// TIA Portal project "SWNC MK2" (V16)

(* hardware
DEVICE "S7-1200 station_1"  S7-1200 Station
   slot 0: "Rack_0"  S7-1200 Rack  Rack  V1.0
   slot 1: "RSF_PLC_Rupert"  CPU 1214C DC/DC/DC  6ES7 214-1AG40-0XB0  V4.4
   slot 2: "DI 8x24VDC_1"  6ES7 221-1BF32-0XB0  V2.0
   slot 3: "CB 1241 (RS485)"  CB 1241 (RS485)  6ES7 241-1CH30-1XB0  V1.0
   slot 3: "DQ 8xRelay_1"  SM 1222 DQ8 x relay  6ES7 222-1HF32-0XB0  V2.0
   slot 4: "AI 8x13BIT_1"  6ES7 231-4HF32-0XB0  V2.1
   slot 5: "AQ 2x14BIT_1"  SM 1232 AQ2  6ES7 232-4HB32-0XB0  V2.1
*)

// ===== PLC "RSF_PLC_Rupert"  CPU 1214C DC/DC/DC =====

VAR_GLOBAL   // PLC tag table "Default tag table"
   "System_Byte" AT %MB1000 : Byte;
   "FirstScan" AT %M1000.0 : Bool;
   "DiagStatusUpdate" AT %M1000.1 : Bool;
   "AlwaysTRUE" AT %M1000.2 : Bool;
   "AlwaysFALSE" AT %M1000.3 : Bool;
   "Clock_Byte" AT %MB1001 : Byte;
   "Clock_10Hz" AT %M1001.0 : Bool;
   "Clock_5Hz" AT %M1001.1 : Bool;
   "Clock_2.5Hz" AT %M1001.2 : Bool;
   "Clock_2Hz" AT %M1001.3 : Bool;
   "Clock_1.25Hz" AT %M1001.4 : Bool;
   "Clock_1Hz" AT %M1001.5 : Bool;
   "Clock_0.625Hz" AT %M1001.6 : Bool;
   "Clock_0.5Hz" AT %M1001.7 : Bool;
   "Mode Bit" AT %MB0 : USInt;
   "HOA Off" AT %M1.0 : Bool;
   "HOA Manual" AT %M1.1 : Bool;
   "HOA Auto Run" AT %M1.2 : Bool;
   "Outside Fan" AT %M1.3 : Bool;
   "Inside Fan" AT %M1.4 : Bool;
   "Outside Cooling" AT %M1.5 : Bool;
   "Inside Cooling" AT %M1.6 : Bool;
   "pump out supply" AT %M1.7 : Bool;
   "pump out Chiller" AT %M2.0 : Bool;
   "pump out inside tank" AT %M2.1 : Bool;
   "Pump out outside tank" AT %M2.2 : Bool;
   "pump out purge tank" AT %M2.3 : Bool;
   "pump chiller circulation" AT %M2.4 : Bool;
   "valve from supply" AT %M2.5 : Bool;   // 0 = to outdoor 1= to indoor
   "valve from chiller" AT %M2.6 : Bool;   // 0 = to outdoor 1= to indoor
   "valve from inside" AT %M2.7 : Bool;   // 0 = to purge 1= to chiller
   "valve from outside" AT %M3.0 : Bool;   // 0 = to purge 1= to chiller
   "chiller enable" AT %M3.1 : Bool;
   "SB OUTSIDE COOLING" AT %M3.2 : Bool;
   "SB INSIDE COOLING" AT %M3.3 : Bool;
   "SB pump out supply" AT %M3.4 : Bool;
   "SB pump out Chiller" AT %M3.5 : Bool;
   "SB pump out inside tank" AT %M3.6 : Bool;
   "SB Pump out outside tank" AT %M3.7 : Bool;
   "SB pump out purge tank" AT %M4.0 : Bool;
   "SB pump chiller circulation" AT %M4.1 : Bool;
   "SB valve from supply" AT %M4.2 : Bool;
   "SB valve from chiller" AT %M4.3 : Bool;
   "SB valve from inside" AT %M4.4 : Bool;
   "SB valve from outside" AT %M4.5 : Bool;
   "SB chiller enable" AT %M4.6 : Bool;
   "SB INSIDE FAN" AT %M4.7 : Bool;
   "SB OUTSIDE FAN" AT %M5.0 : Bool;
   "inside change bit" AT %M5.1 : Bool;   // true when tank change is in progress
   "PB_chill to regen trans" AT %M5.2 : Bool;
   "PB_regen to chill trans" AT %M5.3 : Bool;
END_VAR

VAR_GLOBAL   // PLC tag table "level sensors"
   "supply empty" AT %M0.0 : Bool;
   "chiller full" AT %M0.1 : Bool;
   "chiller empty" AT %M0.2 : Bool;
   "inside full" AT %M0.3 : Bool;
   "inside discharge" AT %M0.4 : Bool;
   "inside empty" AT %M0.5 : Bool;
   "outside full" AT %M0.6 : Bool;
   "outside discharge" AT %M0.7 : Bool;
   "outside empty" AT %M10.0 : Bool;
   "purge full" AT %M10.1 : Bool;
   "purge empty" AT %M10.2 : Bool;
END_VAR

DATA_BLOCK "System Properties"   // DB1
{ S7_Optimized_Access := 'TRUE' }
VERSION : 0.1
   VAR
      "Time" : Struct
         "Current Time" : Time_Of_Day;
         "Night time start" : Time_Of_Day := TOD#20:00:00;
         "Night time end" : Time_Of_Day := TOD#06:00:00;
         "is it day???" : Bool;   // 1 = day, 0 = night
      END_STRUCT;
      "Situation Bits" : Struct
         HOA : Int;
         "Day Run" : Bool;
         "Night Run" : Bool;
         "Day Tank Change" : Int;
         "Night Regen Complete" : Bool;
         "Day/Night Transition Bit" : Int;   // 0= no trans 1= day to night 2= night to day
         "regen or chill" : Int;   // 0 = chill , 1 = regen 3 = transition in progress
         "chilling to regen transition" : Bool;
         "regen to chilling transition" : Bool;
      END_STRUCT;
   END_VAR
BEGIN
END_DATA_BLOCK

DATA_BLOCK "Outputs"   // DB2
{ S7_Optimized_Access := 'TRUE' }
VERSION : 0.1
   VAR
      Fans : Struct
         "Inside Fan" : Bool;
         "Outside Fan" : Bool;
      END_STRUCT;
      "Cooling Pad Pumps" : Struct
         "Inside Cooling" : Bool;
         "Outside Cooling" : Bool;
      END_STRUCT;
      Pumps : Struct
         "From Supply Tank" : Bool;
         "From Chiller Tank" : Bool;
         "From Inside Tank" : Bool;
         "From Outside Tank" : Bool;
         "From Purge Tank" : Bool;
         "Chiller Recirculation" : Bool;
      END_STRUCT;
      Valves : Struct
         "From Supply" : Bool;   // 0= to outdoor, 1= to indoor
         "From Chiller" : Bool;   // 0= to outdoor, 1= to indoor
         "From Indoor" : Bool;   // 0= to Purge, 1= to Chiller
         "From Outdoor" : Bool;   // 0= to Purge, 1= to Chiller
      END_STRUCT;
      Chiller : Struct
         "Chiller Enable" : Bool;
      END_STRUCT;
   END_VAR
BEGIN
END_DATA_BLOCK

DATA_BLOCK "Alarm Conditions"   // DB3
{ S7_Optimized_Access := 'TRUE' }
VERSION : 0.1
   VAR
      "E Stop Pushed" : Bool;
      "Pump Over run" : Bool;
      "Alarm bit" : Bool;
      "Alarm Reset" : Bool;
   END_VAR
BEGIN
END_DATA_BLOCK

DATA_BLOCK "What Time is it?_DB"   // DB4
{ S7_Optimized_Access := 'TRUE' }
VERSION : 0.1
// stored: InstanceOfName What Time is it?
"What Time is it?"
BEGIN
END_DATA_BLOCK

DATA_BLOCK "What mode_DB"   // DB5
{ S7_Optimized_Access := 'TRUE' }
VERSION : 0.1
// stored: InstanceOfName What mode
"What mode"
BEGIN
END_DATA_BLOCK

DATA_BLOCK "Manual Mode_DB"   // DB6
{ S7_Optimized_Access := 'TRUE' }
VERSION : 0.1
// stored: InstanceOfName Manual Mode
"Manual Mode"
BEGIN
END_DATA_BLOCK

DATA_BLOCK "Day Operation_DB"   // DB7
{ S7_Optimized_Access := 'TRUE' }
VERSION : 0.1
// stored: InstanceOfName Day Operation
"Day Operation"
BEGIN
END_DATA_BLOCK

DATA_BLOCK "Night Operation_DB"   // DB8
{ S7_Optimized_Access := 'TRUE' }
VERSION : 0.1
// stored: InstanceOfName Night Operation
"Night Operation"
BEGIN
END_DATA_BLOCK

DATA_BLOCK "Tank check_DB"   // DB9
{ S7_Optimized_Access := 'TRUE' }
VERSION : 0.1
// stored: InstanceOfName Tank check
"Tank check"
BEGIN
END_DATA_BLOCK

DATA_BLOCK "inside tank switch_DB"   // DB11
{ S7_Optimized_Access := 'TRUE' }
VERSION : 0.1
// stored: InstanceOfName inside tank switch
"inside tank switch"
BEGIN
END_DATA_BLOCK

DATA_BLOCK "Auto Run Program_DB"   // DB12
{ S7_Optimized_Access := 'TRUE' }
VERSION : 0.1
// stored: InstanceOfName Auto Run Program
"Auto Run Program"
BEGIN
END_DATA_BLOCK

DATA_BLOCK "Day to Night change_DB"   // DB13
{ S7_Optimized_Access := 'TRUE' }
VERSION : 0.1
// stored: InstanceOfName Day to Night change
"Day to Night change"
BEGIN
END_DATA_BLOCK

DATA_BLOCK "Night to Day change_DB"   // DB14
{ S7_Optimized_Access := 'TRUE' }
VERSION : 0.1
// stored: InstanceOfName Night to Day change
"Night to Day change"
BEGIN
END_DATA_BLOCK

DATA_BLOCK "check for regen transitions_DB"   // DB18
{ S7_Optimized_Access := 'TRUE' }
VERSION : 0.1
// stored: InstanceOfName check for regen transitions
"check for regen transitions"
BEGIN
END_DATA_BLOCK

DATA_BLOCK "chilling to regeneration trans_DB"   // DB19
{ S7_Optimized_Access := 'TRUE' }
VERSION : 0.1
// stored: InstanceOfName chilling to regeneration trans
"chilling to regeneration trans"
BEGIN
END_DATA_BLOCK

DATA_BLOCK "regeneration to chilling trans_DB"   // DB21
{ S7_Optimized_Access := 'TRUE' }
VERSION : 0.1
// stored: InstanceOfName regeneration to chilling trans
"regeneration to chilling trans"
BEGIN
END_DATA_BLOCK

// folder: System blocks/Program resources

DATA_BLOCK "IEC_Timer_0_DB"   // DB10
{ S7_Optimized_Access := 'TRUE' }
AUTHOR : Simatic
FAMILY : IEC
NAME : IEC_TMR
VERSION : 1.0
// stored: InstanceOfName IEC_TIMER
"IEC_TIMER"
BEGIN
END_DATA_BLOCK

DATA_BLOCK "IEC_Timer_0_DB_1"   // DB15
{ S7_Optimized_Access := 'TRUE' }
AUTHOR : Simatic
FAMILY : IEC
NAME : IEC_TMR
VERSION : 1.0
// stored: InstanceOfName IEC_TIMER
"IEC_TIMER"
BEGIN
END_DATA_BLOCK

DATA_BLOCK "IEC_Timer_0_DB_2"   // DB16
{ S7_Optimized_Access := 'TRUE' }
AUTHOR : Simatic
FAMILY : IEC
NAME : IEC_TMR
VERSION : 1.0
// stored: InstanceOfName IEC_TIMER
"IEC_TIMER"
BEGIN
END_DATA_BLOCK

DATA_BLOCK "IEC_Timer_0_DB_3"   // DB17
{ S7_Optimized_Access := 'TRUE' }
AUTHOR : Simatic
FAMILY : IEC
NAME : IEC_TMR
VERSION : 1.0
// stored: InstanceOfName IEC_TIMER
"IEC_TIMER"
BEGIN
END_DATA_BLOCK

DATA_BLOCK "IEC_Timer_0_DB_4"   // DB20
{ S7_Optimized_Access := 'TRUE' }
AUTHOR : Simatic
FAMILY : IEC
NAME : IEC_TMR
VERSION : 1.0
// stored: InstanceOfName IEC_TIMER
"IEC_TIMER"
BEGIN
END_DATA_BLOCK

// folder: (top level)

FUNCTION_BLOCK "What Time is it?"   // FB1, FBD
{ S7_Optimized_Access := 'TRUE' }
VERSION : 0.1
   VAR
      temp1 : DTL;
      OS1 : Bool;
      OS2 : Bool;
      LTNE : Bool;
   END_VAR
   VAR_TEMP
      temp2 : Int;
   END_VAR
   VAR_TEMP   // added for the SCL form of the ladder/FBD networks
      _w1 : Bool;
      _w2 : Bool;
      _w3 : Bool;
   END_VAR
BEGIN

REGION Network 1
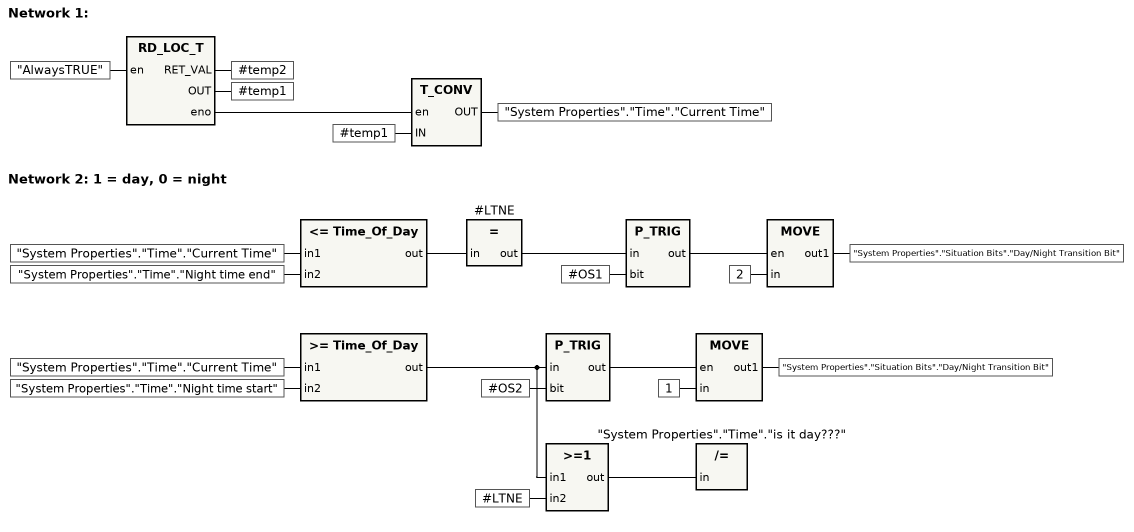
   // ENO of a box is taken as its EN; it also drops when the box reports an error
   #_w1 := "AlwaysTRUE";
   IF #_w1 THEN
       #temp2 := RD_LOC_T(OUT => #temp1);
       "System Properties"."Time"."Current Time" := T_CONV(IN := #temp1);
   END_IF;
END_REGION

REGION Network 2: 1 = day, 0 = night
   // also set the day/night transition integer
   // 0 = no transition
   // 1 = day to night transition
   // 2 = night to day transition
   #LTNE := "System Properties"."Time"."Current Time" <= "System Properties"."Time"."Night time end";
   #_w1 := #LTNE AND NOT #OS1;   // rising edge
   #OS1 := #LTNE;
   IF #_w1 THEN "System Properties"."Situation Bits"."Day/Night Transition Bit" := 2; END_IF;
   #_w2 := "System Properties"."Time"."Current Time" >= "System Properties"."Time"."Night time start";
   #_w3 := #_w2 AND NOT #OS2;   // rising edge
   #OS2 := #_w2;
   IF #_w3 THEN "System Properties"."Situation Bits"."Day/Night Transition Bit" := 1; END_IF;
   "System Properties"."Time"."is it day???" := NOT (#_w2 OR #LTNE);
END_REGION
END_FUNCTION_BLOCK

FUNCTION_BLOCK "What mode"   // FB2, LAD
{ S7_Optimized_Access := 'TRUE' }
VERSION : 0.1
BEGIN

REGION Network 1: Mode selection
   // 0 = startup
   // 1 = off
   // 2 = manual control
   // 3 = automatic run
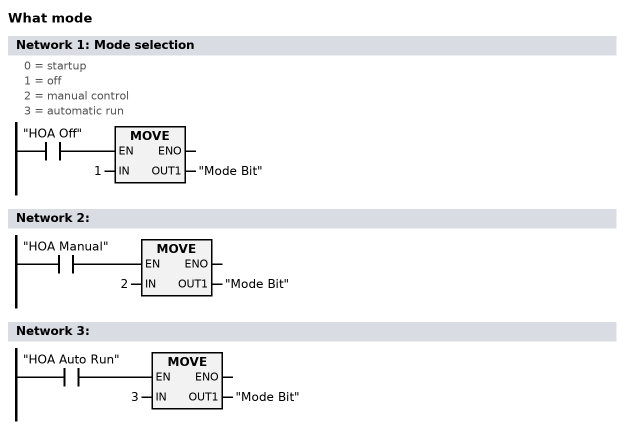
   RUNG wire#powerrail
      Contact( "HOA Off" )
      Move(in := 1, out1 => "Mode Bit")
   END_RUNG
   // the same network as SCL:
   IF "HOA Off" THEN "Mode Bit" := 1; END_IF;
END_REGION

REGION Network 2
   RUNG wire#powerrail
      Contact( "HOA Manual" )
      Move(in := 2, out1 => "Mode Bit")
   END_RUNG
   // the same network as SCL:
   IF "HOA Manual" THEN "Mode Bit" := 2; END_IF;
END_REGION

REGION Network 3
   RUNG wire#powerrail
      Contact( "HOA Auto Run" )
      Move(in := 3, out1 => "Mode Bit")
   END_RUNG
   // the same network as SCL:
   IF "HOA Auto Run" THEN "Mode Bit" := 3; END_IF;
END_REGION
END_FUNCTION_BLOCK

FUNCTION_BLOCK "Manual Mode"   // FB3, LAD
{ S7_Optimized_Access := 'TRUE' }
VERSION : 0.1
BEGIN

REGION Network 1: Manual operation of outputs
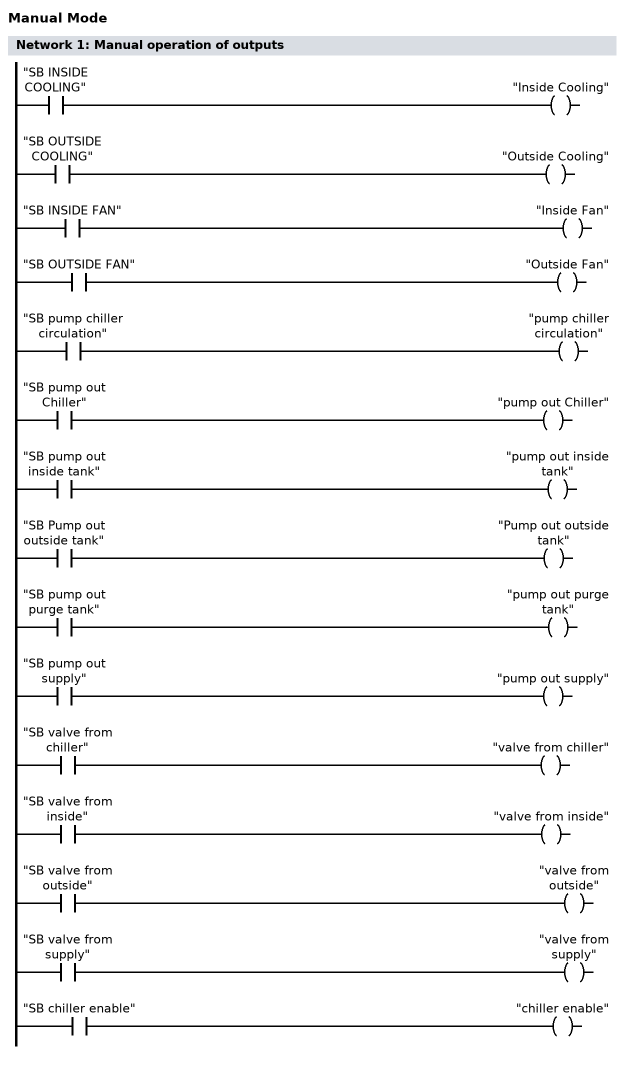
   RUNG wire#powerrail
      Contact( "SB INSIDE COOLING" )
      Coil( "Inside Cooling" )
   END_RUNG
   RUNG wire#powerrail
      Contact( "SB OUTSIDE COOLING" )
      Coil( "Outside Cooling" )
   END_RUNG
   RUNG wire#powerrail
      Contact( "SB INSIDE FAN" )
      Coil( "Inside Fan" )
   END_RUNG
   RUNG wire#powerrail
      Contact( "SB OUTSIDE FAN" )
      Coil( "Outside Fan" )
   END_RUNG
   RUNG wire#powerrail
      Contact( "SB pump chiller circulation" )
      Coil( "pump chiller circulation" )
   END_RUNG
   RUNG wire#powerrail
      Contact( "SB pump out Chiller" )
      Coil( "pump out Chiller" )
   END_RUNG
   RUNG wire#powerrail
      Contact( "SB pump out inside tank" )
      Coil( "pump out inside tank" )
   END_RUNG
   RUNG wire#powerrail
      Contact( "SB Pump out outside tank" )
      Coil( "Pump out outside tank" )
   END_RUNG
   RUNG wire#powerrail
      Contact( "SB pump out purge tank" )
      Coil( "pump out purge tank" )
   END_RUNG
   RUNG wire#powerrail
      Contact( "SB pump out supply" )
      Coil( "pump out supply" )
   END_RUNG
   RUNG wire#powerrail
      Contact( "SB valve from chiller" )
      Coil( "valve from chiller" )
   END_RUNG
   RUNG wire#powerrail
      Contact( "SB valve from inside" )
      Coil( "valve from inside" )
   END_RUNG
   RUNG wire#powerrail
      Contact( "SB valve from outside" )
      Coil( "valve from outside" )
   END_RUNG
   RUNG wire#powerrail
      Contact( "SB valve from supply" )
      Coil( "valve from supply" )
   END_RUNG
   RUNG wire#powerrail
      Contact( "SB chiller enable" )
      Coil( "chiller enable" )
   END_RUNG
   // the same network as SCL:
   "Inside Cooling" := "SB INSIDE COOLING";
   "Outside Cooling" := "SB OUTSIDE COOLING";
   "Inside Fan" := "SB INSIDE FAN";
   "Outside Fan" := "SB OUTSIDE FAN";
   "pump chiller circulation" := "SB pump chiller circulation";
   "pump out Chiller" := "SB pump out Chiller";
   "pump out inside tank" := "SB pump out inside tank";
   "Pump out outside tank" := "SB Pump out outside tank";
   "pump out purge tank" := "SB pump out purge tank";
   "pump out supply" := "SB pump out supply";
   "valve from chiller" := "SB valve from chiller";
   "valve from inside" := "SB valve from inside";
   "valve from outside" := "SB valve from outside";
   "valve from supply" := "SB valve from supply";
   "chiller enable" := "SB chiller enable";
END_REGION
END_FUNCTION_BLOCK

FUNCTION_BLOCK "Auto Run Program"   // FB4, LAD
{ S7_Optimized_Access := 'TRUE' }
VERSION : 0.1
BEGIN

REGION Network 1: Select for day or night operation
   // only works when there is not transitions happening
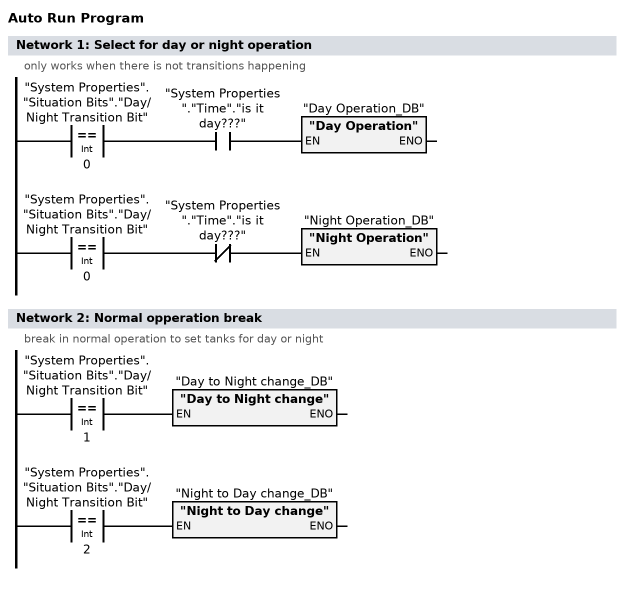
   RUNG wire#powerrail
      { S7_Templates := "SrcType := Int" } EQ_Contact(in1 := "System Properties"."Situation Bits"."Day/Night Transition Bit", in2 := 0)
      Contact( "System Properties"."Time"."is it day???" )
      "Day Operation_DB"()
   END_RUNG
   RUNG wire#powerrail
      { S7_Templates := "SrcType := Int" } EQ_Contact(in1 := "System Properties"."Situation Bits"."Day/Night Transition Bit", in2 := 0)
      I_Contact( "System Properties"."Time"."is it day???" )
      "Night Operation_DB"()
   END_RUNG
   // the same network as SCL:
   IF ("System Properties"."Situation Bits"."Day/Night Transition Bit" = 0) AND "System Properties"."Time"."is it day???" THEN
       "Day Operation_DB"();   // "Day Operation"
   END_IF;
   IF ("System Properties"."Situation Bits"."Day/Night Transition Bit" = 0) AND NOT "System Properties"."Time"."is it day???" THEN
       "Night Operation_DB"();   // "Night Operation"
   END_IF;
END_REGION

REGION Network 2: Normal opperation break
   // break in normal operation to set tanks for day or night
   RUNG wire#powerrail
      { S7_Templates := "SrcType := Int" } EQ_Contact(in1 := "System Properties"."Situation Bits"."Day/Night Transition Bit", in2 := 1)
      "Day to Night change_DB"()
   END_RUNG
   RUNG wire#powerrail
      { S7_Templates := "SrcType := Int" } EQ_Contact(in1 := "System Properties"."Situation Bits"."Day/Night Transition Bit", in2 := 2)
      "Night to Day change_DB"()
   END_RUNG
   // the same network as SCL:
   IF "System Properties"."Situation Bits"."Day/Night Transition Bit" = 1 THEN
       "Day to Night change_DB"();   // "Day to Night change"
   END_IF;
   IF "System Properties"."Situation Bits"."Day/Night Transition Bit" = 2 THEN
       "Night to Day change_DB"();   // "Night to Day change"
   END_IF;
END_REGION
END_FUNCTION_BLOCK

FUNCTION_BLOCK "Day Operation"   // FB5, LAD
{ S7_Optimized_Access := 'TRUE' }
VERSION : 0.1
   VAR_TEMP   // added for the SCL form of the ladder/FBD networks
      _w1 : Bool;
   END_VAR
BEGIN

REGION Network 1: Place Holder
   // to make VFD control
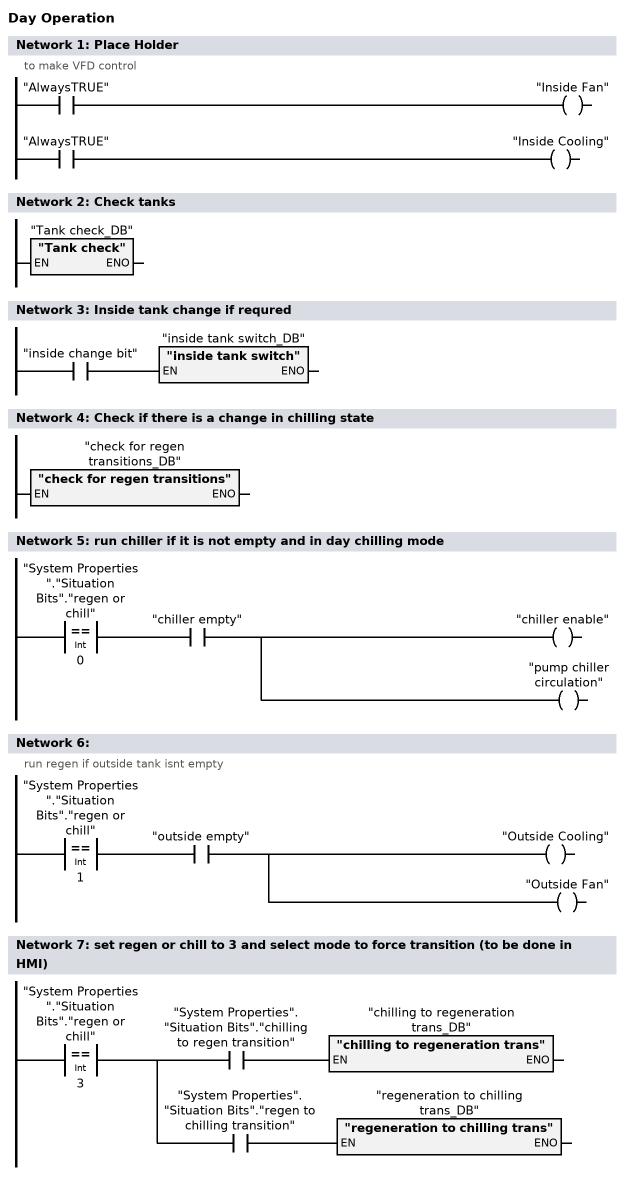
   RUNG wire#powerrail
      Contact( "AlwaysTRUE" )
      Coil( "Inside Fan" )
   END_RUNG
   RUNG wire#powerrail
      Contact( "AlwaysTRUE" )
      Coil( "Inside Cooling" )
   END_RUNG
   // the same network as SCL:
   "Inside Fan" := "AlwaysTRUE";
   "Inside Cooling" := "AlwaysTRUE";
END_REGION

REGION Network 2: Check tanks
   RUNG wire#powerrail
      "Tank check_DB"()
   END_RUNG
   // the same network as SCL:
   "Tank check_DB"();   // "Tank check"
END_REGION

REGION Network 3: Inside tank change if requred
   RUNG wire#powerrail
      Contact( "inside change bit" )
      "inside tank switch_DB"()
   END_RUNG
   // the same network as SCL:
   IF "inside change bit" THEN
       "inside tank switch_DB"();   // "inside tank switch"
   END_IF;
END_REGION

REGION Network 4: Check if there is a change in chilling state
   RUNG wire#powerrail
      "check for regen transitions_DB"()
   END_RUNG
   // the same network as SCL:
   "check for regen transitions_DB"();   // "check for regen transitions"
END_REGION

REGION Network 5: run chiller if it is not empty and in day chilling mode
   RUNG wire#powerrail
      { S7_Templates := "SrcType := Int" } EQ_Contact(in1 := "System Properties"."Situation Bits"."regen or chill", in2 := 0)
      Contact( "chiller empty" )
      wire#w1
      Coil( "chiller enable" )
   END_RUNG
   RUNG wire#w1
      Coil( "pump chiller circulation" )
   END_RUNG
   // the same network as SCL:
   "chiller enable" := ("System Properties"."Situation Bits"."regen or chill" = 0) AND "chiller empty";
   "pump chiller circulation" := "chiller enable";
END_REGION

REGION Network 6
   // run regen if outside tank isnt empty
   RUNG wire#powerrail
      { S7_Templates := "SrcType := Int" } EQ_Contact(in1 := "System Properties"."Situation Bits"."regen or chill", in2 := 1)
      Contact( "outside empty" )
      wire#w1
      Coil( "Outside Cooling" )
   END_RUNG
   RUNG wire#w1
      Coil( "Outside Fan" )
   END_RUNG
   // the same network as SCL:
   "Outside Cooling" := ("System Properties"."Situation Bits"."regen or chill" = 1) AND "outside empty";
   "Outside Fan" := "Outside Cooling";
END_REGION

REGION Network 7: set regen or chill to 3 and select mode to force transition (to be done in HMI)
   RUNG wire#powerrail
      { S7_Templates := "SrcType := Int" } EQ_Contact(in1 := "System Properties"."Situation Bits"."regen or chill", in2 := 3)
      wire#w1
      Contact( "System Properties"."Situation Bits"."chilling to regen transition" )
      "chilling to regeneration trans_DB"()
   END_RUNG
   RUNG wire#w1
      Contact( "System Properties"."Situation Bits"."regen to chilling transition" )
      "regeneration to chilling trans_DB"()
   END_RUNG
   // the same network as SCL:
   #_w1 := "System Properties"."Situation Bits"."regen or chill" = 3;
   IF #_w1 AND "System Properties"."Situation Bits"."chilling to regen transition" THEN
       "chilling to regeneration trans_DB"();   // "chilling to regeneration trans"
   END_IF;
   IF #_w1 AND "System Properties"."Situation Bits"."regen to chilling transition" THEN
       "regeneration to chilling trans_DB"();   // "regeneration to chilling trans"
   END_IF;
END_REGION
END_FUNCTION_BLOCK

FUNCTION_BLOCK "Night Operation"   // FB6, LAD
{ S7_Optimized_Access := 'TRUE' }
VERSION : 0.1
BEGIN

REGION Network 1
   // place holder will be VFD
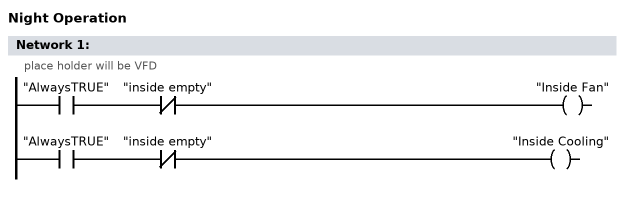
   RUNG wire#powerrail
      Contact( "AlwaysTRUE" )
      I_Contact( "inside empty" )
      Coil( "Inside Fan" )
   END_RUNG
   RUNG wire#powerrail
      Contact( "AlwaysTRUE" )
      I_Contact( "inside empty" )
      Coil( "Inside Cooling" )
   END_RUNG
   // the same network as SCL:
   "Inside Fan" := "AlwaysTRUE" AND NOT "inside empty";
   "Inside Cooling" := "AlwaysTRUE" AND NOT "inside empty";
END_REGION
END_FUNCTION_BLOCK

FUNCTION_BLOCK "Tank check"   // FB7, LAD
{ S7_Optimized_Access := 'TRUE' }
VERSION : 0.1
BEGIN

REGION Network 1: sets to true when the inside tank hits its discharge level
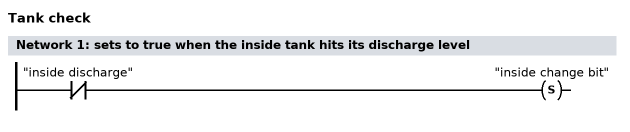
   RUNG wire#powerrail
      I_Contact( "inside discharge" )
      S_Coil( "inside change bit" )
   END_RUNG
   // the same network as SCL:
   IF NOT "inside discharge" THEN "inside change bit" := TRUE; END_IF;
END_REGION
END_FUNCTION_BLOCK

FUNCTION_BLOCK "inside tank switch"   // FB8, LAD
{ S7_Optimized_Access := 'TRUE' }
VERSION : 0.1
   VAR_TEMP   // added for the SCL form of the ladder/FBD networks
      _w1 : Bool;
   END_VAR
BEGIN

REGION Network 1: valve set up --- 0 = to purge 1= to chiller
   // set to purge (valve is not energised)
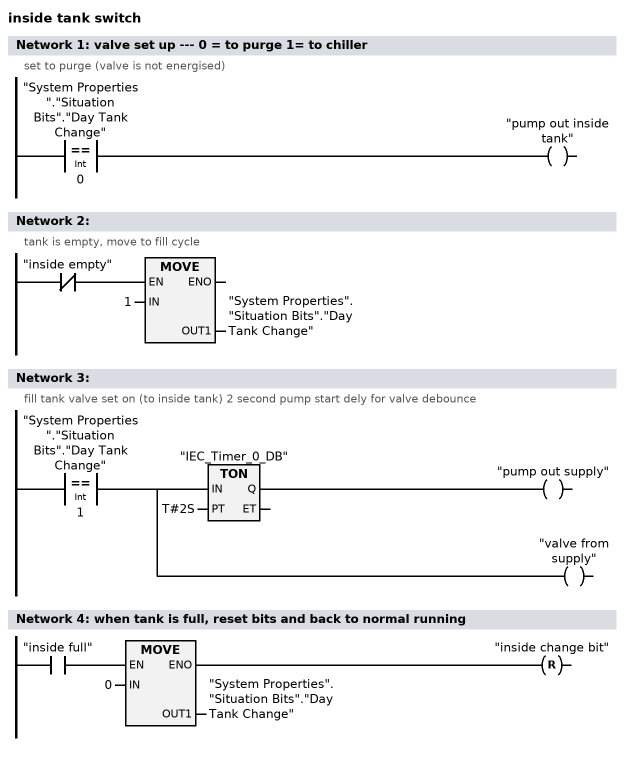
   RUNG wire#powerrail
      { S7_Templates := "SrcType := Int" } EQ_Contact(in1 := "System Properties"."Situation Bits"."Day Tank Change", in2 := 0)
      Coil( "pump out inside tank" )
   END_RUNG
   // the same network as SCL:
   "pump out inside tank" := "System Properties"."Situation Bits"."Day Tank Change" = 0;
END_REGION

REGION Network 2
   // tank is empty, move to fill cycle
   RUNG wire#powerrail
      I_Contact( "inside empty" )
      Move(in := 1, out1 => "System Properties"."Situation Bits"."Day Tank Change")
   END_RUNG
   // the same network as SCL:
   IF NOT "inside empty" THEN "System Properties"."Situation Bits"."Day Tank Change" := 1; END_IF;
END_REGION

REGION Network 3
   // fill tank valve set on (to inside tank) 2 second pump start dely for valve debounce
   #_w1 := "System Properties"."Situation Bits"."Day Tank Change" = 1;
   "IEC_Timer_0_DB".TON(IN := #_w1, PT := T#2S);
   "pump out supply" := "IEC_Timer_0_DB".Q;
   "valve from supply" := #_w1;
END_REGION

REGION Network 4: when tank is full, reset bits and back to normal running
   RUNG wire#powerrail
      Contact( "inside full" )
      Move(in := 0, out1 => "System Properties"."Situation Bits"."Day Tank Change")
      R_Coil( "inside change bit" )
   END_RUNG
   // the same network as SCL:
   IF "inside full" THEN
       "System Properties"."Situation Bits"."Day Tank Change" := 0;
       "inside change bit" := FALSE;
   END_IF;
END_REGION
END_FUNCTION_BLOCK

FUNCTION_BLOCK "Day to Night change"   // FB9, LAD
{ S7_Optimized_Access := 'TRUE' }
VERSION : 0.1
   VAR
      "DN change bit" : Int;
   END_VAR
   VAR_TEMP   // added for the SCL form of the ladder/FBD networks
      _w1 : Bool;
   END_VAR
BEGIN

REGION Network 1
   // inside tank to purge (valve at 0)
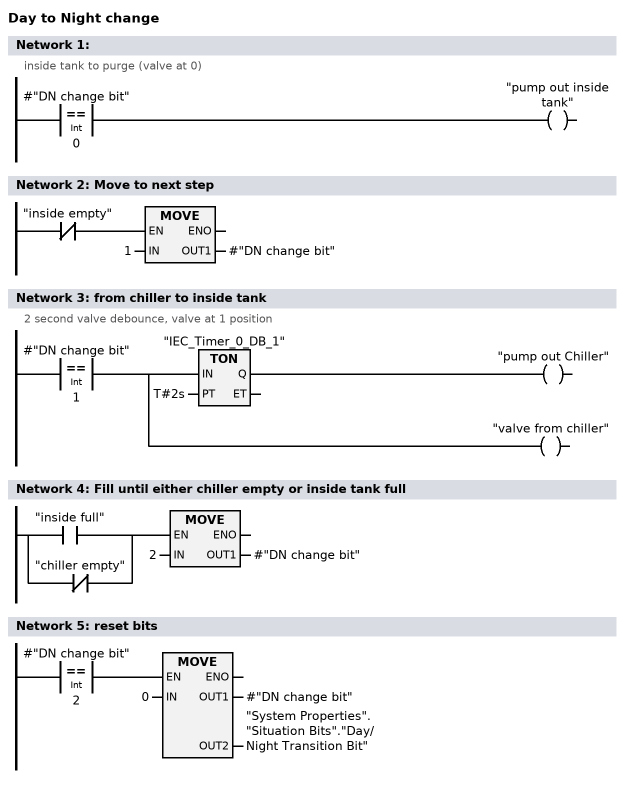
   RUNG wire#powerrail
      { S7_Templates := "SrcType := Int" } EQ_Contact(in1 := #"DN change bit", in2 := 0)
      Coil( "pump out inside tank" )
   END_RUNG
   // the same network as SCL:
   "pump out inside tank" := #"DN change bit" = 0;
END_REGION

REGION Network 2: Move to next step
   RUNG wire#powerrail
      I_Contact( "inside empty" )
      Move(in := 1, out1 => #"DN change bit")
   END_RUNG
   // the same network as SCL:
   IF NOT "inside empty" THEN #"DN change bit" := 1; END_IF;
END_REGION

REGION Network 3: from chiller to inside tank
   // 2 second valve debounce, valve at 1 position
   #_w1 := #"DN change bit" = 1;
   "IEC_Timer_0_DB_1".TON(IN := #_w1, PT := T#2s);
   "pump out Chiller" := "IEC_Timer_0_DB_1".Q;
   "valve from chiller" := #_w1;
END_REGION

REGION Network 4: Fill until either chiller empty or inside tank full
   RUNG wire#powerrail
      Contact( "inside full" )
      wire#w1
      Move(in := 2, out1 => #"DN change bit")
   END_RUNG
   RUNG wire#powerrail
      I_Contact( "chiller empty" )
   END_RUNG wire#w1
   // the same network as SCL:
   IF "inside full" OR NOT "chiller empty" THEN #"DN change bit" := 2; END_IF;
END_REGION

REGION Network 5: reset bits
   RUNG wire#powerrail
      { S7_Templates := "SrcType := Int" } EQ_Contact(in1 := #"DN change bit", in2 := 2)
      Move(in := 0, out1 => #"DN change bit", out2 => "System Properties"."Situation Bits"."Day/Night Transition Bit")
   END_RUNG
   // the same network as SCL:
   IF #"DN change bit" = 2 THEN
       #"DN change bit" := 0;
       "System Properties"."Situation Bits"."Day/Night Transition Bit" := 0;
   END_IF;
END_REGION
END_FUNCTION_BLOCK

FUNCTION_BLOCK "Night to Day change"   // FB10, LAD
{ S7_Optimized_Access := 'TRUE' }
VERSION : 0.1
   VAR
      "ND change bit" : Int;
   END_VAR
   VAR_TEMP   // added for the SCL form of the ladder/FBD networks
      _w1 : Bool;
   END_VAR
BEGIN

REGION Network 1: move from inside back to chiller
   // 2 second valve debounce
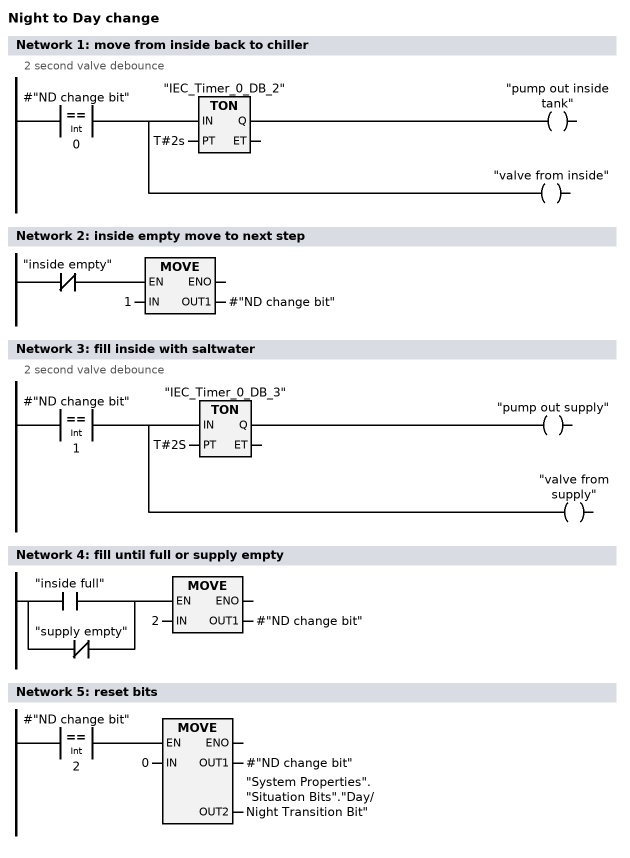
   #_w1 := #"ND change bit" = 0;
   "IEC_Timer_0_DB_2".TON(IN := #_w1, PT := T#2s);
   "pump out inside tank" := "IEC_Timer_0_DB_2".Q;
   "valve from inside" := #_w1;
END_REGION

REGION Network 2: inside empty move to next step
   RUNG wire#powerrail
      I_Contact( "inside empty" )
      Move(in := 1, out1 => #"ND change bit")
   END_RUNG
   // the same network as SCL:
   IF NOT "inside empty" THEN #"ND change bit" := 1; END_IF;
END_REGION

REGION Network 3: fill inside with saltwater
   // 2 second valve debounce
   #_w1 := #"ND change bit" = 1;
   "IEC_Timer_0_DB_3".TON(IN := #_w1, PT := T#2S);
   "pump out supply" := "IEC_Timer_0_DB_3".Q;
   "valve from supply" := #_w1;
END_REGION

REGION Network 4: fill until full or supply empty
   RUNG wire#powerrail
      Contact( "inside full" )
      wire#w1
      Move(in := 2, out1 => #"ND change bit")
   END_RUNG
   RUNG wire#powerrail
      I_Contact( "supply empty" )
   END_RUNG wire#w1
   // the same network as SCL:
   IF "inside full" OR NOT "supply empty" THEN #"ND change bit" := 2; END_IF;
END_REGION

REGION Network 5: reset bits
   RUNG wire#powerrail
      { S7_Templates := "SrcType := Int" } EQ_Contact(in1 := #"ND change bit", in2 := 2)
      Move(in := 0, out1 => #"ND change bit", out2 => "System Properties"."Situation Bits"."Day/Night Transition Bit")
   END_RUNG
   // the same network as SCL:
   IF #"ND change bit" = 2 THEN
       #"ND change bit" := 0;
       "System Properties"."Situation Bits"."Day/Night Transition Bit" := 0;
   END_IF;
END_REGION
END_FUNCTION_BLOCK

FUNCTION_BLOCK "check for regen transitions"   // FB11, LAD
{ S7_Optimized_Access := 'TRUE' }
VERSION : 0.1
   VAR
      OS3 : Bool;
      OS4 : Bool;
   END_VAR
   VAR_TEMP   // added for the SCL form of the ladder/FBD networks
      _w1 : Bool;
   END_VAR
BEGIN

REGION Network 1
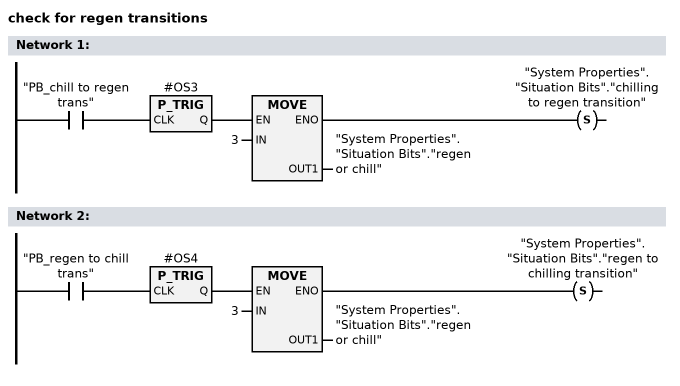
   RUNG wire#powerrail
      Contact( "PB_chill to regen trans" )
      P_Trig( #OS3 )
      Move(in := 3, out1 => "System Properties"."Situation Bits"."regen or chill")
      S_Coil( "System Properties"."Situation Bits"."chilling to regen transition" )
   END_RUNG
   // the same network as SCL:
   #_w1 := "PB_chill to regen trans" AND NOT #OS3;   // rising edge
   #OS3 := "PB_chill to regen trans";
   IF #_w1 THEN
       "System Properties"."Situation Bits"."regen or chill" := 3;
       "System Properties"."Situation Bits"."chilling to regen transition" := TRUE;
   END_IF;
END_REGION

REGION Network 2
   RUNG wire#powerrail
      Contact( "PB_regen to chill trans" )
      P_Trig( #OS4 )
      Move(in := 3, out1 => "System Properties"."Situation Bits"."regen or chill")
      S_Coil( "System Properties"."Situation Bits"."regen to chilling transition" )
   END_RUNG
   // the same network as SCL:
   #_w1 := "PB_regen to chill trans" AND NOT #OS4;   // rising edge
   #OS4 := "PB_regen to chill trans";
   IF #_w1 THEN
       "System Properties"."Situation Bits"."regen or chill" := 3;
       "System Properties"."Situation Bits"."regen to chilling transition" := TRUE;
   END_IF;
END_REGION
END_FUNCTION_BLOCK

FUNCTION_BLOCK "chilling to regeneration trans"   // FB12, LAD
{ S7_Optimized_Access := 'TRUE' }
VERSION : 0.1
   VAR
      "internal bit" : Int;
   END_VAR
   VAR_TEMP   // added for the SCL form of the ladder/FBD networks
      _w1 : Bool;
   END_VAR
BEGIN

REGION Network 1: make sure outside is empty
   // valve in position 0 to purge
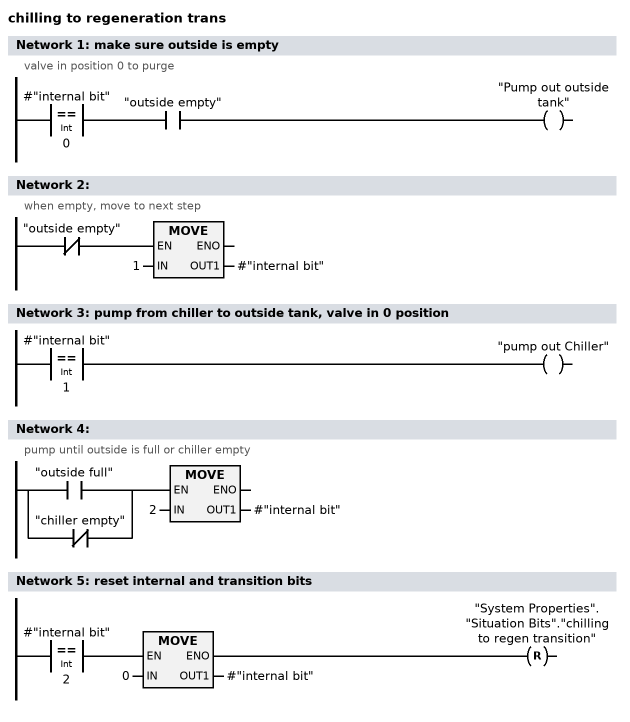
   RUNG wire#powerrail
      { S7_Templates := "SrcType := Int" } EQ_Contact(in1 := #"internal bit", in2 := 0)
      Contact( "outside empty" )
      Coil( "Pump out outside tank" )
   END_RUNG
   // the same network as SCL:
   "Pump out outside tank" := (#"internal bit" = 0) AND "outside empty";
END_REGION

REGION Network 2
   // when empty, move to next step
   RUNG wire#powerrail
      I_Contact( "outside empty" )
      Move(in := 1, out1 => #"internal bit")
   END_RUNG
   // the same network as SCL:
   IF NOT "outside empty" THEN #"internal bit" := 1; END_IF;
END_REGION

REGION Network 3: pump from chiller to outside tank, valve in 0 position
   RUNG wire#powerrail
      { S7_Templates := "SrcType := Int" } EQ_Contact(in1 := #"internal bit", in2 := 1)
      Coil( "pump out Chiller" )
   END_RUNG
   // the same network as SCL:
   "pump out Chiller" := #"internal bit" = 1;
END_REGION

REGION Network 4
   // pump until outside is full or chiller empty
   RUNG wire#powerrail
      Contact( "outside full" )
      wire#w1
      Move(in := 2, out1 => #"internal bit")
   END_RUNG
   RUNG wire#powerrail
      I_Contact( "chiller empty" )
   END_RUNG wire#w1
   // the same network as SCL:
   IF "outside full" OR NOT "chiller empty" THEN #"internal bit" := 2; END_IF;
END_REGION

REGION Network 5: reset internal and transition bits
   RUNG wire#powerrail
      { S7_Templates := "SrcType := Int" } EQ_Contact(in1 := #"internal bit", in2 := 2)
      Move(in := 0, out1 => #"internal bit")
      R_Coil( "System Properties"."Situation Bits"."chilling to regen transition" )
   END_RUNG
   // the same network as SCL:
   #_w1 := #"internal bit" = 2;
   IF #_w1 THEN
       #"internal bit" := 0;
       "System Properties"."Situation Bits"."chilling to regen transition" := FALSE;
   END_IF;
END_REGION
END_FUNCTION_BLOCK

FUNCTION_BLOCK "regeneration to chilling trans"   // FB13, LAD
{ S7_Optimized_Access := 'TRUE' }
VERSION : 0.1
   VAR
      "internal bit" : Int;
   END_VAR
   VAR_TEMP   // added for the SCL form of the ladder/FBD networks
      _w1 : Bool;
   END_VAR
BEGIN

REGION Network 1: empty outside tank to chiller
   // 2 second valve debounce
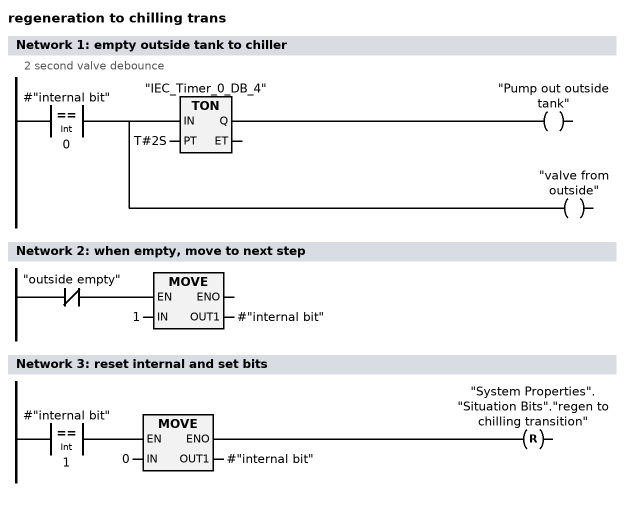
   #_w1 := #"internal bit" = 0;
   "IEC_Timer_0_DB_4".TON(IN := #_w1, PT := T#2S);
   "Pump out outside tank" := "IEC_Timer_0_DB_4".Q;
   "valve from outside" := #_w1;
END_REGION

REGION Network 2: when empty, move to next step
   RUNG wire#powerrail
      I_Contact( "outside empty" )
      Move(in := 1, out1 => #"internal bit")
   END_RUNG
   // the same network as SCL:
   IF NOT "outside empty" THEN #"internal bit" := 1; END_IF;
END_REGION

REGION Network 3: reset internal and set bits
   RUNG wire#powerrail
      { S7_Templates := "SrcType := Int" } EQ_Contact(in1 := #"internal bit", in2 := 1)
      Move(in := 0, out1 => #"internal bit")
      R_Coil( "System Properties"."Situation Bits"."regen to chilling transition" )
   END_RUNG
   // the same network as SCL:
   #_w1 := #"internal bit" = 1;
   IF #_w1 THEN
       #"internal bit" := 0;
       "System Properties"."Situation Bits"."regen to chilling transition" := FALSE;
   END_IF;
END_REGION
END_FUNCTION_BLOCK

ORGANIZATION_BLOCK "Main"   // OB1, LAD, ProgramCycle
TITLE = "Main Program Sweep (Cycle)"
{ S7_Optimized_Access := 'TRUE' }
VERSION : 0.1
   VAR_INPUT
      Initial_Call : Bool;   // Initial call of this OB
      Remanence : Bool;   // =True, if remanent data are available
   END_VAR
   VAR_TEMP
      placeholder : Bool;
   END_VAR
BEGIN

REGION Network 1: Work out if it's day or night
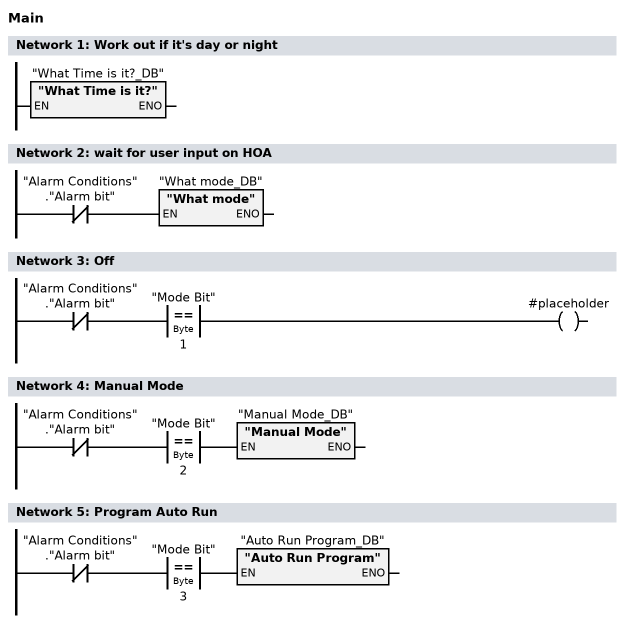
   RUNG wire#powerrail
      "What Time is it?_DB"()
   END_RUNG
   // the same network as SCL:
   "What Time is it?_DB"();   // "What Time is it?"
END_REGION

REGION Network 2: wait for user input on HOA
   RUNG wire#powerrail
      I_Contact( "Alarm Conditions"."Alarm bit" )
      "What mode_DB"()
   END_RUNG
   // the same network as SCL:
   IF NOT "Alarm Conditions"."Alarm bit" THEN
       "What mode_DB"();   // "What mode"
   END_IF;
END_REGION

REGION Network 3: Off
   RUNG wire#powerrail
      I_Contact( "Alarm Conditions"."Alarm bit" )
      { S7_Templates := "SrcType := Byte" } EQ_Contact(in1 := "Mode Bit", in2 := 1)
      Coil( #placeholder )
   END_RUNG
   // the same network as SCL:
   #placeholder := NOT "Alarm Conditions"."Alarm bit" AND ("Mode Bit" = 1);
END_REGION

REGION Network 4: Manual Mode
   RUNG wire#powerrail
      I_Contact( "Alarm Conditions"."Alarm bit" )
      { S7_Templates := "SrcType := Byte" } EQ_Contact(in1 := "Mode Bit", in2 := 2)
      "Manual Mode_DB"()
   END_RUNG
   // the same network as SCL:
   IF NOT "Alarm Conditions"."Alarm bit" AND ("Mode Bit" = 2) THEN
       "Manual Mode_DB"();   // "Manual Mode"
   END_IF;
END_REGION

REGION Network 5: Program Auto Run
   RUNG wire#powerrail
      I_Contact( "Alarm Conditions"."Alarm bit" )
      { S7_Templates := "SrcType := Byte" } EQ_Contact(in1 := "Mode Bit", in2 := 3)
      "Auto Run Program_DB"()
   END_RUNG
   // the same network as SCL:
   IF NOT "Alarm Conditions"."Alarm bit" AND ("Mode Bit" = 3) THEN
       "Auto Run Program_DB"();   // "Auto Run Program"
   END_IF;
END_REGION
END_ORGANIZATION_BLOCK

ORGANIZATION_BLOCK "Startup"   // OB100, LAD, Startup
TITLE = "Complete Restart"
{ S7_Optimized_Access := 'TRUE' }
VERSION : 0.1
   VAR_INPUT
      LostRetentive : Bool;   // True if retentive data are lost
      LostRTC : Bool;   // True if date and time are lost
   END_VAR
   VAR_TEMP
      temp1 : Int;
      temp2 : Int;
   END_VAR
BEGIN

REGION Network 1: Put Program In Start Up Mode (0) and ensure sub program set bits are 0
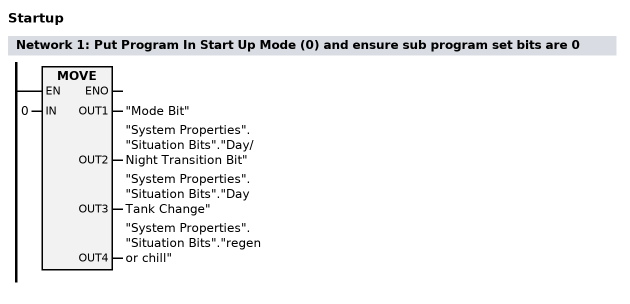
   RUNG wire#powerrail
      Move(in := 0, out1 => "Mode Bit", out2 => "System Properties"."Situation Bits"."Day/Night Transition Bit", out3 => "System Properties"."Situation Bits"."Day Tank Change", out4 => "System Properties"."Situation Bits"."regen or chill")
   END_RUNG
   // the same network as SCL:
   "Mode Bit" := 0;
   "System Properties"."Situation Bits"."Day/Night Transition Bit" := 0;
   "System Properties"."Situation Bits"."Day Tank Change" := 0;
   "System Properties"."Situation Bits"."regen or chill" := 0;
END_REGION
END_ORGANIZATION_BLOCK